// TIA Portal V18 export
// export: Created 2026-06-22T15:41:33.8809672Z, ExportSetting WithDefaults, DisplayName Totally Integrated Automation Portal, DisplayVersion V18, DisplayName TIA Portal Openness, DisplayVersion V18, DisplayName TIA Portal Version Control Interface, DisplayVersion V18, DisplayName STEP 7 Professional, DisplayVersion V18, DisplayName STEP 7 Safety, DisplayVersion V18, DisplayName WinCC Professional, DisplayVersion V18
DATA_BLOCK "DB11_GuiSangPLC2"   // DB11
{ S7_Optimized_Access := 'FALSE' }
VERSION : 0.1
// stored: AutoNumber true, IsOnlyStoredInLoadMemory false, IsWriteProtectedInAS false
   VAR
      Speed_SP_toSend : Real;
      Control_Byte_toSend : Bool;
      Reset_Cmd_toSend : Bool;
      DIR_Cmd_toSend : Bool;
   END_VAR
BEGIN
END_DATA_BLOCK
